FUNCTION_BLOCK Eventos_PLC 
VAR_INPUT
	bResetArrayAvisos:BOOL;
	bClearEvents:BOOL;
END_VAR
VAR_OUTPUT
END_VAR
VAR
	fbMessage : FB_TcMessage;
	fbAlarm : FB_TcAlarm;
	fbTcEventLogger: FB_TcEventLogger;
    ITcClearLoggedEventsSettings : I_TcClearLoggedEventsSettings;
	fbAdsReadEvents:FB_AdsReadEvents;
	ArrayAvisos:ARRAY [1..100] OF BOOL;
	ArrayAlarmas:ARRAY [1..100] OF BOOL;
	i:INT;
	FalloPrueba:BOOL;
	bReadEvent: BOOL;
	//Prueba
    bReadEvents          : BOOL;
    bClear               : BOOL;
END_VAR

//Llamadas de funciones 
Llamadas_Y_funciones();

//  >>>>>>>>>>>>>>>>>>>>>>>>>>>>>>>>>>>>> Avisos <<<<<<<<<<<<<<<<<<<<<<<<<<<<<<<<<<<<<<<<<<
//Los avisos solo son a modo informativo. 




//Aviso 1        Lectura a PLC a maestro deshabilitada
IF NOT MAIN_Orden_Lectura_PLCs.bHabilitaLectura_Maestro AND NOT ArrayAvisos[1] THEN 
	ArrayAvisos[1]:=TRUE;
	fbMessage.CreateEx(TC_Events.My_Events.Lectura_PLC_Maestro_deshabilitada, 0);
	SendAviso();
END_IF
//Aviso 2        Lectura a PLCs deshabilitada
IF NOT MAIN_Orden_Lectura_PLCs.bHabilitarLecturaDePLCs AND NOT ArrayAvisos[2] THEN 
	ArrayAvisos[2]:=TRUE;
	fbMessage.CreateEx(TC_Events.My_Events.LecturaPLCsDeshabilitada, 0);
	SendAviso();
END_IF


//  >>>>>>>>>>>>>>>>>>>>>>>>>>>>>>>>>>>>> Alarmas <<<<<<<<<<<<<<<<<<<<<<<<<<<<<<<<<<<<<<<<<<
//Son fallos críticos. 

//Alarma 1  Fallo comunicación con PLC Maestro
 IF Lectura_Maestro.fbLectura_a_PLC_Maestro.AlarmaFalloComunicacion  AND NOT ArrayAlarmas[1] THEN 
	ArrayAlarmas[1]:=TRUE;
	fbAlarm.CreateEx(TC_Events.My_Events.FalloLecturaPLC_Maestro, FALSE ,0);
	SendAlarma();
END_IF

//Alarma 2 Prueba 
IF FalloPrueba AND NOT ArrayAlarmas[2] THEN 
	ArrayAlarmas[2]:=TRUE;
	fbAlarm.CreateEx(TC_EVENTS.My_Events.Prueba,FALSE,0);
	SendAlarma();
END_IF

{warning 'add method implementation '}
METHOD BorraEventos : BOOL
fbTcEventLogger.ClearLoggedEvents(ipClearSettings:= ITcClearLoggedEventsSettings);
END_METHOD

ACTION Llamadas_Y_funciones:
//Reset array de los avisos    <<<<<<<<<<<<<<<   utilizados para que solo se envíe un mensaje y no esté continuamente enviando 
IF bResetArrayAvisos THEN 
	ResetArrayEvents();
END_IF

//Borrar avisos del HMI 
IF bClearEvents THEN 
	BorraEventos();
	ResetArrayEvents();
END_IF
END_ACTION

{warning 'add method implementation '}
METHOD ResetArrayEvents : BOOL
FOR i := 1 TO 100 BY 1 DO 
	ArrayAvisos[i]:= FALSE;
	ArrayAlarmas[i]:=FALSE;
END_FOR
END_METHOD

{warning 'add method implementation '}
METHOD SendAlarma : BOOL
fbAlarm.Raise(0);
END_METHOD

{warning 'add method implementation '}
METHOD SendAviso : BOOL
fbMessage.Send(0);
END_METHOD

END_FUNCTION_BLOCK

(* stored: Version 1.1.0.1, ProductVersion 3.1.4024.12
   POU Eventos_PLC: Id {98e2f037-c32c-4c67-8faa-8f8fcffc9bcf}, SpecialFunc None
   Method BorraEventos: Id {f5274ab3-21ca-4503-b70c-058d78dea58e}
   Action Llamadas_Y_funciones: Id {87bab000-2c8c-4caf-886b-ce6b2d9f5f18}
   Method ResetArrayEvents: Id {30ab97c2-6826-44d9-ad0b-d9aad256c76d}
   Method SendAlarma: Id {fdb62939-b029-4f72-a768-915bbf038581}
   Method SendAviso: Id {ecc7c34c-76c7-48bd-90b5-fffa4044d2f0} *)
